FUNCTION_BLOCK Test_TStreamAdd_Read_Short_STRING EXTENDS TUnitTestBase
VAR
    Stream : TStream(StreamLength := 2);
    TestString : STRING(10) := '0123456789';
END_VAR



Stream.Init(2);

Stream.Add_STRING(TestString);
    
Assertion.AssertEquals_UDINT(
    Expected := 11,
    Actual := Stream.Position,
    VariableName := 'Stream.Position');
    
Stream.Add_DINT(12345678);

Assertion.AssertEquals_UDINT(
    Expected := 15,
    Actual := Stream.Position,
    VariableName := 'Stream.Position');
    
Stream.Seek(0);

Assertion.AssertEquals_STRING(
    Expected := TestString,
    Actual := Stream.Read_STRING(),
    VariableName := 'Stream.Read_STRING()');
    
Assertion.AssertEquals_UDINT(
    Expected := 11,
    Actual := Stream.Position,
    VariableName := 'Stream.Position');
    
Assertion.AssertEquals_UDINT(
    Expected := 12345678,
    Actual := Stream.Read_UDINT(),
    VariableName := 'Stream.Read_UDINT()');



TestFinished();

END_FUNCTION_BLOCK

(* stored: Version 1.1.0.1, ProductVersion 3.1.4024.4
   POU Test_TStreamAdd_Read_Short_STRING: Id {9ca0ea26-0b16-4608-9d44-cef6e71d8a4a}, SpecialFunc None *)
